Staubli VAL3: Form_PanelBool.pgx

public program Form_PanelBool(string x_sTitle, string x_sPanelTitle, bool& x_bList[], num& x_nSelectIndex, string x_sBottom, string x_sYes, string x_sNo)
  local num l_nNum
begin

//×××××××××××××××××××××××××××××××××××××××××××××××××
//×××××××××××××××××××××××××××××××××××××××××××××××××
resize(sBuff,1,size(x_bList))
for l_nNum=0 to size(x_bList)-1
  if x_bList[l_nNum]
    sBuff[l_nNum]=toString("",l_nNum+1)+"."+x_sYes
  else
    sBuff[l_nNum]=toString("",l_nNum+1)+"."+x_sNo
  endIf
endFor
//*************************************************
call Form_PanelList(x_sTitle,x_sPanelTitle,sBuff,x_nSelectIndex,x_sBottom)



end
